// TIA Portal V16 export
// export: Created 2022-04-06T03:32:48.3247043Z, ExportSetting WithDefaults, DisplayName Totally Integrated Automation Portal, DisplayVersion V16 Update 4, DisplayName TIA Portal Version Control Interface, DisplayVersion V16 Update 2, DisplayName TIA Portal Openness, DisplayVersion V16 Update 4, DisplayName SINAMICS Startdrive Advanced, DisplayVersion V16, DisplayName SINAMICS Startdrive G130, G150, S120, S150, SINAMICS MV, S210, DisplayVersion V16, DisplayName SINAMICS Startdrive G110M, G120, G120C, G120D, G120P, DisplayVersion V16, DisplayName STEP 7 Professional, DisplayVersion V16 Update 4, DisplayName STEP 7 Safety, DisplayVersion V16, DisplayName WinCC Professional, DisplayVersion V16 Update 4
FUNCTION_BLOCK "fbAlarmedSetpoint"   // FB6, LAD
{ S7_Optimized_Access := 'TRUE' }
VERSION : 0.1
// Processes raw analog input and evaluates alarms.
// Note: All alarms are momentary, i.e. no ack necessary and they reset themselves when the condition becomes false.
// stored: AutoNumber true, IsIECCheckEnabled false, IsRetainMemResEnabled false, MemoryReserve 100, SetENOAutomatically false, UDAEnableTagReadback false
   VAR_INPUT
      iInRawValue { ExternalAccessible := 'False'; ExternalVisible := 'False'; ExternalWritable := 'False'} : Real;
   END_VAR
   VAR RETAIN
      arrSetpoints { ExternalVisible := 'False'} : Array[1..10] of "udtTimeOfDaySetpoint";   // Setpoints need to be chronologically increasing
      rSetpoint { ExternalVisible := 'False'; ExternalWritable := 'False'} : Real;
      rActual { ExternalVisible := 'False'; ExternalWritable := 'False'} : Real;
      Alarms { ExternalVisible := 'False'; ExternalWritable := 'False'} : Struct
         bHigh { ExternalVisible := 'False'; ExternalWritable := 'False'} : Bool;   // rActual exceeds limit
         bLow { ExternalVisible := 'False'; ExternalWritable := 'False'} : Bool;   // rActual exceeds limit
         bRate { ExternalVisible := 'False'; ExternalWritable := 'False'} : Bool;   // rActual increases or decreases faster than the limit. False if rate is left as 0.
         bSetpoint { ExternalVisible := 'False'; ExternalWritable := 'False'} : Bool;   // rActual does not reach rSetpoint within allowed time delay and deadband. False if deadband left at 0.
      END_STRUCT;
      Config { ExternalVisible := 'False'} : Struct
         rLowCalibration { ExternalVisible := 'False'} : Real := 0.0;
         rHighCalibration { ExternalVisible := 'False'} : Real := 100.0;
         Alarms { ExternalVisible := 'False'} : Struct
            rLowLimit { ExternalVisible := 'False'} : Real := 0.0;
            rHighLimit { ExternalVisible := 'False'} : Real := 100.0;
            rRateLimit { ExternalVisible := 'False'} : Real;   // Maximum permitted change in rActual per second
            rDeadband { ExternalVisible := 'False'} : Real;   // Range around rSetpoint that is still considered within range
            iSettlingSecs { ExternalVisible := 'False'} : Int;   // Allowable delay to allow rActual to reach rSetpoint after change
         END_STRUCT;
      END_STRUCT;
   END_VAR
   VAR
      TON_RateCheck { ExternalAccessible := 'False'; ExternalVisible := 'False'; ExternalWritable := 'False'} : TON_TIME;
      rActual_Prev { ExternalAccessible := 'False'; ExternalVisible := 'False'; ExternalWritable := 'False'} : Real;
      TON_Settling { ExternalAccessible := 'False'; ExternalVisible := 'False'; ExternalWritable := 'False'} : TON_TIME;
      rSetpoint_Prev { ExternalAccessible := 'False'; ExternalVisible := 'False'; ExternalWritable := 'False'} : Real;
   END_VAR
   VAR_TEMP
      localTime : Date_And_Time;
      ret_val : Int;
      currentTOD : Time_Of_Day;
      i : Int;
      currentTODsecs : DInt;
   END_VAR
   VAR_TEMP   // added for the SCL form of the ladder/FBD networks
      _w1 : Bool;
      _w2 : Bool;
   END_VAR
BEGIN

REGION Network 1 (SCL): Scale raw input based on calibration
   #rActual := #iInRawValue;
   //"fcAnalogInput"(iInRawValue := #iInRawValue,
   //                           rLowCalibration := #Config.rLowCalibration,
   //                            rHighCalibration := #Config.rHighCalibration);
END_REGION

REGION Network 2 (SCL): Low/high alarms
   #Alarms.bHigh := #rActual > #Config.Alarms.rHighLimit;
   #Alarms.bLow  := #rActual < #Config.Alarms.rLowLimit;
END_REGION

REGION Network 3 (SCL): Rate of change alarm
   // Set the current value on startup to prevent a spurious alarm
   IF "FirstScan" THEN
       #rActual_Prev := #rActual;
   END_IF;

   // Compare values at every given time interval to get rate of change
   IF #TON_RateCheck.Q THEN
       #Alarms.bRate := ( ABS(#rActual - #rActual_Prev) > #Config.Alarms.rRateLimit)
       AND (#Config.Alarms.rRateLimit <> 0.0); // ignore alarm if max rate is left at default of 0

       #rActual_Prev := #rActual;
   END_IF;

   #TON_RateCheck(IN := NOT #TON_RateCheck.Q,
                  PT := t#1s);
END_REGION

REGION Network 4: Get current time of day
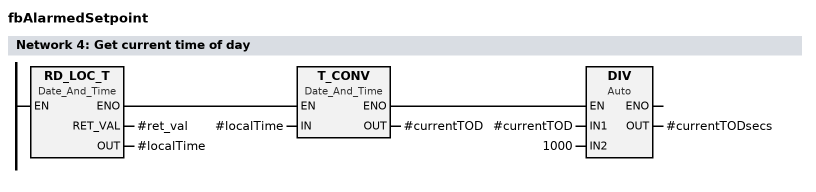
   RUNG wire#powerrail
      { S7_Templates := "date_type := Date_And_Time" } RD_LOC_T(RET_VAL => #ret_val, OUT => #localTime)
      { S7_Templates := "[src_type := Date_And_Time, dest_type := Time_Of_Day]" } T_CONV(IN := #localTime, OUT => #currentTOD)
      Div(in1 := #currentTOD, in2 := 1000, out => #currentTODsecs)
   END_RUNG
   // the same network as SCL:
   #ret_val := RD_LOC_T(OUT => #localTime, ENO => #_w1);
   T_CONV(EN := #_w1, IN := #localTime, OUT => #currentTOD, ENO => #_w2);
   IF #_w2 THEN #currentTODsecs := #currentTOD / 1000; END_IF;
END_REGION

REGION Network 5 (SCL): Determine current setpoint based on time of day
   IF #arrSetpoints[1].TimeOfDaySeconds = -1 THEN
       // If no time schedule is defined, default to first setpoint in array
       #rSetpoint := #arrSetpoints[1].rSetpoint;

   ELSIF #currentTODsecs < #arrSetpoints[1].TimeOfDaySeconds THEN
       // Check for setpoint from previous day
       FOR #i := 10 TO 1 BY -1 DO
           IF #arrSetpoints[#i].TimeOfDaySeconds <> -1 THEN
               #rSetpoint := #arrSetpoints[#i].rSetpoint;
               EXIT;
           END_IF;
       END_FOR;

   ELSE
       // Iterate through and find current setpoint
       FOR #i := 1 TO 9 DO
           IF #currentTODsecs < #arrSetpoints[#i + 1].TimeOfDaySeconds OR #arrSetpoints[#i + 1].TimeOfDaySeconds = -1 THEN
               #rSetpoint := #arrSetpoints[#i].rSetpoint;
               EXIT;
           ELSIF #i = 9 THEN
               #rSetpoint := #arrSetpoints[10].rSetpoint;
           END_IF;
       END_FOR;

   END_IF;
END_REGION

REGION Network 6 (SCL): Setpoint not reached alarm


   // Set the current value on startup to prevent a spurious alarm
   IF "FirstScan" THEN
       #rSetpoint_Prev := #rSetpoint;
   END_IF;

   // Evaluate alarm after settling time has elapsed
   #TON_Settling(IN := (#rSetpoint = #rSetpoint_Prev), // restart timer when setpoint changes
                 PT := INT_TO_TIME(#Config.Alarms.iSettlingSecs * 1000)); // convert to ms

   #Alarms.bSetpoint := #TON_Settling.Q AND (
   (#rActual < #rSetpoint - #Config.Alarms.rDeadband / 2.0) OR
   (#rActual > #rSetpoint + #Config.Alarms.rDeadband / 2.0) )
   AND (#Config.Alarms.rDeadband <> 0.0); // ignore alarm if deadband is left at default of 0

   // Save setpoint value for next comparison
   #rSetpoint_Prev := #rSetpoint;
END_REGION
END_FUNCTION_BLOCK
